ABB RAPID module: Module1.mod

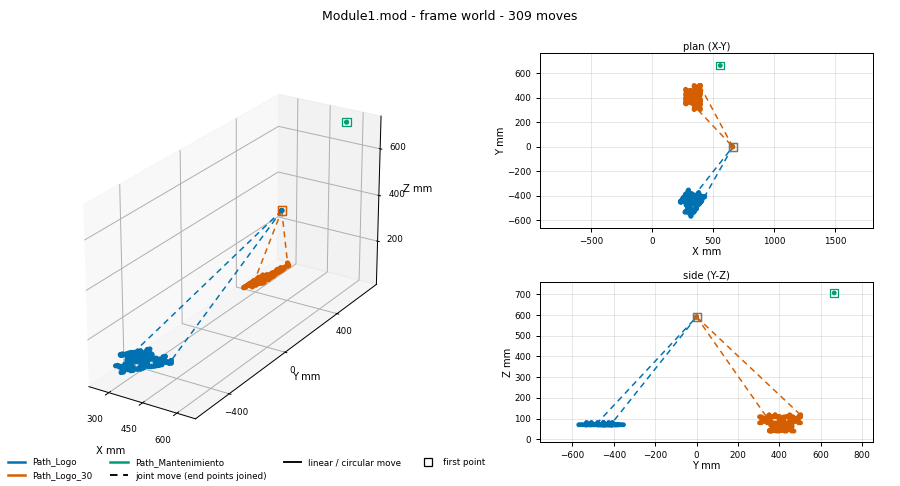
[picture p0: tool path of Module1.mod in frame world, 309 of 309 moves have a stored position in this frame; points joined in program order, loops and branches not executed]
MODULE Module1
        PERS tooldata TToolLab1:=[TRUE,[[120.208,0,145.208],[0.923879533,0,0.382683432,0]],[0.1,[47.87,0,69.665],[1,0,0,0],0,0,0]];
    TASK PERS wobjdata Logo:=[FALSE,TRUE,"",[[0,0,0],[1,0,0,0]],[[400,-450,60],[0.30070845,0,0,0.953716115]]];
    TASK PERS wobjdata Logo30:=[FALSE,TRUE,"",[[0,0,0],[1,0,0,0]],[[400,450,100],[0,-0.258819045,0,0.965925826]]];
    CONST robtarget Inicio:=[[44.962359667,-517.867347375,530.792],[0.115076142,0.881118798,0.277818382,-0.364971357],[0,0,-1,1],[9E+09,9E+09,9E+09,9E+09,9E+09,9E+09]];
    CONST robtarget X1_offset:=[[0,-52.582,20],[0,0,1,0],[-1,-3,-1,1],[9E+09,9E+09,9E+09,9E+09,9E+09,9E+09]];
    CONST robtarget Target_10:=[[0,-52.582,10],[0,0,1,0],[-1,-3,-1,1],[9E+09,9E+09,9E+09,9E+09,9E+09,9E+09]];
    CONST robtarget Target_20:=[[14.731,-43.214,10],[0,0,1,0],[-1,-3,-1,1],[9E+09,9E+09,9E+09,9E+09,9E+09,9E+09]];
    CONST robtarget Target_30:=[[29.461,-33.847,10],[0,0,1,0],[-1,-3,-1,1],[9E+09,9E+09,9E+09,9E+09,9E+09,9E+09]];
    CONST robtarget Target_40:=[[44.144,-42.928,10],[0,0,1,0],[-1,-3,-1,1],[9E+09,9E+09,9E+09,9E+09,9E+09,9E+09]];
    CONST robtarget Target_50:=[[58.827,-52.009,10],[0,0,1,0],[-1,-3,-1,1],[9E+09,9E+09,9E+09,9E+09,9E+09,9E+09]];
    CONST robtarget Target_60:=[[58.827,-43.047,10],[0,0,1,0],[-1,-3,-1,1],[9E+09,9E+09,9E+09,9E+09,9E+09,9E+09]];
    CONST robtarget Target_70:=[[47.314,-36.04,10],[0,0,1,0],[-1,-3,-1,1],[9E+09,9E+09,9E+09,9E+09,9E+09,9E+09]];
    CONST robtarget Target_80:=[[35.801,-29.032,10],[0,0,1,0],[-1,-3,-1,1],[9E+09,9E+09,9E+09,9E+09,9E+09,9E+09]];
    CONST robtarget Target_90:=[[47.314,-21.881,10],[0,0,1,0],[-1,-3,-1,1],[9E+09,9E+09,9E+09,9E+09,9E+09,9E+09]];
    CONST robtarget Target_100:=[[58.827,-14.73,10],[0,0,1,0],[-1,-3,-1,1],[9E+09,9E+09,9E+09,9E+09,9E+09,9E+09]];
    CONST robtarget Target_110:=[[58.827,-6.293,10],[0,0,1,0],[-1,-3,-1,1],[9E+09,9E+09,9E+09,9E+09,9E+09,9E+09]];
    CONST robtarget Target_120:=[[44.334,-15.493,10],[0,0,1,0],[-1,-3,-1,1],[9E+09,9E+09,9E+09,9E+09,9E+09,9E+09]];
    CONST robtarget Target_130:=[[29.842,-24.694,10],[0,0,1,0],[-1,-3,-1,1],[9E+09,9E+09,9E+09,9E+09,9E+09,9E+09]];
    CONST robtarget Target_140:=[[14.921,-15.493,10],[0,0,1,0],[-1,-3,-1,1],[9E+09,9E+09,9E+09,9E+09,9E+09,9E+09]];
    CONST robtarget Target_150:=[[0,-6.293,10],[0,0,1,0],[-1,-3,-1,1],[9E+09,9E+09,9E+09,9E+09,9E+09,9E+09]];
    CONST robtarget Target_160:=[[0,-15.255,10],[0,0,1,0],[-1,-3,-1,1],[9E+09,9E+09,9E+09,9E+09,9E+09,9E+09]];
    CONST robtarget Target_170:=[[11.727,-22.406,10],[0,0,1,0],[-1,-3,-1,1],[9E+09,9E+09,9E+09,9E+09,9E+09,9E+09]];
    CONST robtarget Target_180:=[[23.455,-29.556,10],[0,0,1,0],[-1,-3,-1,1],[9E+09,9E+09,9E+09,9E+09,9E+09,9E+09]];
    CONST robtarget Target_190:=[[11.727,-36.85,10],[0,0,1,0],[-1,-3,-1,1],[9E+09,9E+09,9E+09,9E+09,9E+09,9E+09]];
    CONST robtarget Target_200:=[[0,-44.144,10],[0,0,1,0],[-1,-3,-1,1],[9E+09,9E+09,9E+09,9E+09,9E+09,9E+09]];
    CONST robtarget B_offset:=[[0,0,20],[0,0,1,0],[-1,-3,-1,1],[9E+09,9E+09,9E+09,9E+09,9E+09,9E+09]];
    CONST robtarget Target_210:=[[0.000068234,0,10],[0,0,1,0],[-1,-3,-1,1],[9E+09,9E+09,9E+09,9E+09,9E+09,9E+09]];
    CONST robtarget Target_220:=[[29.413525648,0.000000006,10],[0,0,1,0],[-1,-3,-1,1],[9E+09,9E+09,9E+09,9E+09,9E+09,9E+09]];
    CONST robtarget Target_230:=[[58.826983061,0.000000012,10],[0,0,1,0],[-1,-3,-1,1],[9E+09,9E+09,9E+09,9E+09,9E+09,9E+09]];
    CONST robtarget Target_240:=[[58.826263831,7.794172482,10],[0,0,1,0],[-1,-3,-1,1],[9E+09,9E+09,9E+09,9E+09,9E+09,9E+09]];
    CONST robtarget Target_250:=[[58.826363749,15.588918532,10],[0,0,1,0],[-1,-3,-1,1],[9E+09,9E+09,9E+09,9E+09,9E+09,9E+09]];
    CONST robtarget Target_260:=[[58.421279237,25.027558611,10],[0,0,1,0],[-1,-3,-1,1],[9E+09,9E+09,9E+09,9E+09,9E+09,9E+09]];
    CONST robtarget Target_270:=[[56.442373859,31.03371666,10],[0,0,1,0],[-1,-3,-1,1],[9E+09,9E+09,9E+09,9E+09,9E+09,9E+09]];
    CONST robtarget Target_280:=[[52.032676311,35.682055346,10],[0,0,1,0],[-1,-3,-1,1],[9E+09,9E+09,9E+09,9E+09,9E+09,9E+09]];
    CONST robtarget Target_290:=[[45.573477335,37.136157676,10],[0,0,1,0],[-1,-3,-1,1],[9E+09,9E+09,9E+09,9E+09,9E+09,9E+09]];
    CONST robtarget Target_300:=[[38.136561779,34.942815929,10],[0,0,1,0],[-1,-3,-1,1],[9E+09,9E+09,9E+09,9E+09,9E+09,9E+09]];
    CONST robtarget Target_310:=[[32.98791054,28.888765515,10],[0,0,1,0],[-1,-3,-1,1],[9E+09,9E+09,9E+09,9E+09,9E+09,9E+09]];
    CONST robtarget Target_320:=[[27.482150174,37.016714998,10],[0,0,1,0],[-1,-3,-1,1],[9E+09,9E+09,9E+09,9E+09,9E+09,9E+09]];
    CONST robtarget Target_330:=[[18.067037183,39.901013935,10],[0,0,1,0],[-1,-3,-1,1],[9E+09,9E+09,9E+09,9E+09,9E+09,9E+09]];
    CONST robtarget Target_340:=[[10.320457963,38.231853851,10],[0,0,1,0],[-1,-3,-1,1],[9E+09,9E+09,9E+09,9E+09,9E+09,9E+09]];
    CONST robtarget Target_350:=[[4.766871396,33.798677084,10],[0,0,1,0],[-1,-3,-1,1],[9E+09,9E+09,9E+09,9E+09,9E+09,9E+09]];
    CONST robtarget Target_360:=[[1.096188095,26.671237284,10],[0,0,1,0],[-1,-3,-1,1],[9E+09,9E+09,9E+09,9E+09,9E+09,9E+09]];
    CONST robtarget Target_370:=[[-0.000000003,16.874785035,10],[0,0,1,0],[-1,-3,-1,1],[9E+09,9E+09,9E+09,9E+09,9E+09,9E+09]];
    CONST robtarget Target_380:=[[0.000156899,8.438088883,10],[0,0,1,0],[-1,-3,-1,1],[9E+09,9E+09,9E+09,9E+09,9E+09,9E+09]];
    CONST robtarget O_offset:=[[-1.24,70.315,20],[0,0,1,0],[-1,-3,-1,1],[9E+09,9E+09,9E+09,9E+09,9E+09,9E+09]];
    CONST robtarget Target_390:=[[-1.239782829,70.315479984,10],[0,0,1,0],[-1,-3,-1,1],[9E+09,9E+09,9E+09,9E+09,9E+09,9E+09]];
    CONST robtarget Target_400:=[[0.786338624,59.588668628,10],[0,0,1,0],[-1,-3,-1,1],[9E+09,9E+09,9E+09,9E+09,9E+09,9E+09]];
    CONST robtarget Target_410:=[[6.769482618,51.342081579,10],[0,0,1,0],[-1,-3,-1,1],[9E+09,9E+09,9E+09,9E+09,9E+09,9E+09]];
    CONST robtarget Target_420:=[[16.422507661,46.146190366,10],[0,0,1,0],[-1,-3,-1,1],[9E+09,9E+09,9E+09,9E+09,9E+09,9E+09]];
    CONST robtarget Target_430:=[[29.412921119,44.334619996,10],[0,0,1,0],[-1,-3,-1,1],[9E+09,9E+09,9E+09,9E+09,9E+09,9E+09]];
    CONST robtarget Target_440:=[[42.42730153,46.169208644,10],[0,0,1,0],[-1,-3,-1,1],[9E+09,9E+09,9E+09,9E+09,9E+09,9E+09]];
    CONST robtarget Target_450:=[[52.103968369,51.389690987,10],[0,0,1,0],[-1,-3,-1,1],[9E+09,9E+09,9E+09,9E+09,9E+09,9E+09]];
    CONST robtarget Target_460:=[[58.039423406,59.613427273,10],[0,0,1,0],[-1,-3,-1,1],[9E+09,9E+09,9E+09,9E+09,9E+09,9E+09]];
    CONST robtarget Target_470:=[[60.065636343,70.315019731,10],[0,0,1,0],[-1,-3,-1,1],[9E+09,9E+09,9E+09,9E+09,9E+09,9E+09]];
    CONST robtarget Target_480:=[[57.967982157,81.137015477,10],[0,0,1,0],[-1,-3,-1,1],[9E+09,9E+09,9E+09,9E+09,9E+09,9E+09]];
    CONST robtarget Target_490:=[[52.104377969,89.287851626,10],[0,0,1,0],[-1,-3,-1,1],[9E+09,9E+09,9E+09,9E+09,9E+09,9E+09]];
    CONST robtarget Target_500:=[[42.475192456,94.484565525,10],[0,0,1,0],[-1,-3,-1,1],[9E+09,9E+09,9E+09,9E+09,9E+09,9E+09]];
    CONST robtarget Target_510:=[[29.412679756,96.343313211,10],[0,0,1,0],[-1,-3,-1,1],[9E+09,9E+09,9E+09,9E+09,9E+09,9E+09]];
    CONST robtarget Target_520:=[[16.469896844,94.532001119,10],[0,0,1,0],[-1,-3,-1,1],[9E+09,9E+09,9E+09,9E+09,9E+09,9E+09]];
    CONST robtarget Target_530:=[[6.769065997,89.288494859,10],[0,0,1,0],[-1,-3,-1,1],[9E+09,9E+09,9E+09,9E+09,9E+09,9E+09]];
    CONST robtarget Target_540:=[[0.714522275,80.873942209,10],[0,0,1,0],[-1,-3,-1,1],[9E+09,9E+09,9E+09,9E+09,9E+09,9E+09]];
    CONST robtarget X2_offset:=[[0,99.299,20],[0,0,1,0],[-1,-3,-1,1],[9E+09,9E+09,9E+09,9E+09,9E+09,9E+09]];
    CONST robtarget Target_550:=[[0,99.299,10],[0,0,1,0],[-1,-3,-1,1],[9E+09,9E+09,9E+09,9E+09,9E+09,9E+09]];
    CONST robtarget Target_560:=[[14.73,108.667,10],[0,0,1,0],[-1,-3,-1,1],[9E+09,9E+09,9E+09,9E+09,9E+09,9E+09]];
    CONST robtarget Target_570:=[[29.46,118.034,10],[0,0,1,0],[-1,-3,-1,1],[9E+09,9E+09,9E+09,9E+09,9E+09,9E+09]];
    CONST robtarget Target_580:=[[44.143,108.953,10],[0,0,1,0],[-1,-3,-1,1],[9E+09,9E+09,9E+09,9E+09,9E+09,9E+09]];
    CONST robtarget Target_590:=[[58.826,99.871,10],[0,0,1,0],[-1,-3,-1,1],[9E+09,9E+09,9E+09,9E+09,9E+09,9E+09]];
    CONST robtarget Target_600:=[[58.826,108.834,10],[0,0,1,0],[-1,-3,-1,1],[9E+09,9E+09,9E+09,9E+09,9E+09,9E+09]];
    CONST robtarget Target_610:=[[47.313,115.841,10],[0,0,1,0],[-1,-3,-1,1],[9E+09,9E+09,9E+09,9E+09,9E+09,9E+09]];
    CONST robtarget Target_620:=[[35.801,122.849,10],[0,0,1,0],[-1,-3,-1,1],[9E+09,9E+09,9E+09,9E+09,9E+09,9E+09]];
    CONST robtarget Target_630:=[[47.313,130,10],[0,0,1,0],[-1,-3,-1,1],[9E+09,9E+09,9E+09,9E+09,9E+09,9E+09]];
    CONST robtarget Target_640:=[[58.826,137.15,10],[0,0,1,0],[-1,-3,-1,1],[9E+09,9E+09,9E+09,9E+09,9E+09,9E+09]];
    CONST robtarget Target_650:=[[58.826,145.588,10],[0,0,1,0],[-1,-3,-1,1],[9E+09,9E+09,9E+09,9E+09,9E+09,9E+09]];
    CONST robtarget Target_660:=[[44.334,136.388,10],[0,0,1,0],[-1,-3,-1,1],[9E+09,9E+09,9E+09,9E+09,9E+09,9E+09]];
    CONST robtarget Target_670:=[[29.842,127.187,10],[0,0,1,0],[-1,-3,-1,1],[9E+09,9E+09,9E+09,9E+09,9E+09,9E+09]];
    CONST robtarget Target_680:=[[14.92,136.387,10],[0,0,1,0],[-1,-3,-1,1],[9E+09,9E+09,9E+09,9E+09,9E+09,9E+09]];
    CONST robtarget Target_690:=[[-0.001,145.588,10],[0,0,1,0],[-1,-3,-1,1],[9E+09,9E+09,9E+09,9E+09,9E+09,9E+09]];
    CONST robtarget Target_700:=[[-0.001,136.626,10],[0,0,1,0],[-1,-3,-1,1],[9E+09,9E+09,9E+09,9E+09,9E+09,9E+09]];
    CONST robtarget Target_710:=[[11.726,129.475,10],[0,0,1,0],[-1,-3,-1,1],[9E+09,9E+09,9E+09,9E+09,9E+09,9E+09]];
    CONST robtarget Target_720:=[[23.454,122.324,10],[0,0,1,0],[-1,-3,-1,1],[9E+09,9E+09,9E+09,9E+09,9E+09,9E+09]];
    CONST robtarget Target_730:=[[11.727,115.031,10],[0,0,1,0],[-1,-3,-1,1],[9E+09,9E+09,9E+09,9E+09,9E+09,9E+09]];
    CONST robtarget Target_740:=[[-0.001,107.737,10],[0,0,1,0],[-1,-3,-1,1],[9E+09,9E+09,9E+09,9E+09,9E+09,9E+09]];
    CONST robtarget R_offset:=[[80.066,24.872,20],[0,0,1,0],[-1,-3,-1,1],[9E+09,9E+09,9E+09,9E+09,9E+09,9E+09]];
    CONST robtarget Target_750:=[[80.066,24.872,10],[0,0,1,0],[-1,-3,-1,1],[9E+09,9E+09,9E+09,9E+09,9E+09,9E+09]];
    CONST robtarget Target_760:=[[80.066,17.292,10],[0,0,1,0],[-1,-3,-1,1],[9E+09,9E+09,9E+09,9E+09,9E+09,9E+09]];
    CONST robtarget Target_770:=[[80.066,9.712,10],[0,0,1,0],[-1,-3,-1,1],[9E+09,9E+09,9E+09,9E+09,9E+09,9E+09]];
    CONST robtarget Target_780:=[[80.614,1.251,10],[0,0,1,0],[-1,-3,-1,1],[9E+09,9E+09,9E+09,9E+09,9E+09,9E+09]];
    CONST robtarget Target_790:=[[83.165,-5.256,10],[0,0,1,0],[-1,-3,-1,1],[9E+09,9E+09,9E+09,9E+09,9E+09,9E+09]];
    CONST robtarget Target_800:=[[88.289,-10.143,10],[0,0,1,0],[-1,-3,-1,1],[9E+09,9E+09,9E+09,9E+09,9E+09,9E+09]];
    CONST robtarget Target_810:=[[96.036,-11.93,10],[0,0,1,0],[-1,-3,-1,1],[9E+09,9E+09,9E+09,9E+09,9E+09,9E+09]];
    CONST robtarget Target_820:=[[106.833,-8.641,10],[0,0,1,0],[-1,-3,-1,1],[9E+09,9E+09,9E+09,9E+09,9E+09,9E+09]];
    CONST robtarget Target_830:=[[113.293,0.274,10],[0,0,1,0],[-1,-3,-1,1],[9E+09,9E+09,9E+09,9E+09,9E+09,9E+09]];
    CONST robtarget Target_840:=[[126.093,-10.19,10],[0,0,1,0],[-1,-3,-1,1],[9E+09,9E+09,9E+09,9E+09,9E+09,9E+09]];
    CONST robtarget Target_850:=[[138.892,-20.654,10],[0,0,1,0],[-1,-3,-1,1],[9E+09,9E+09,9E+09,9E+09,9E+09,9E+09]];
    CONST robtarget Target_860:=[[138.892,-10.5,10],[0,0,1,0],[-1,-3,-1,1],[9E+09,9E+09,9E+09,9E+09,9E+09,9E+09]];
    CONST robtarget Target_870:=[[127.189,-1.204,10],[0,0,1,0],[-1,-3,-1,1],[9E+09,9E+09,9E+09,9E+09,9E+09,9E+09]];
    CONST robtarget Target_880:=[[115.486,8.092,10],[0,0,1,0],[-1,-3,-1,1],[9E+09,9E+09,9E+09,9E+09,9E+09,9E+09]];
    CONST robtarget Target_890:=[[115.486,17.054,10],[0,0,1,0],[-1,-3,-1,1],[9E+09,9E+09,9E+09,9E+09,9E+09,9E+09]];
    CONST robtarget Target_900:=[[127.189,17.054,10],[0,0,1,0],[-1,-3,-1,1],[9E+09,9E+09,9E+09,9E+09,9E+09,9E+09]];
    CONST robtarget Target_910:=[[138.892,17.054,10],[0,0,1,0],[-1,-3,-1,1],[9E+09,9E+09,9E+09,9E+09,9E+09,9E+09]];
    CONST robtarget Target_920:=[[138.892,24.872,10],[0,0,1,0],[-1,-3,-1,1],[9E+09,9E+09,9E+09,9E+09,9E+09,9E+09]];
    CONST robtarget Target_930:=[[109.479,24.872,10],[0,0,1,0],[-1,-3,-1,1],[9E+09,9E+09,9E+09,9E+09,9E+09,9E+09]];
    CONST robtarget J1_offset:=[[80.066,56.669,20],[0,0,1,0],[-1,-3,-1,1],[9E+09,9E+09,9E+09,9E+09,9E+09,9E+09]];
    CONST robtarget Target_940:=[[80.066,56.669,10],[0,0,1,0],[-1,-3,-1,1],[9E+09,9E+09,9E+09,9E+09,9E+09,9E+09]];
    CONST robtarget Target_950:=[[80.066,46.538,10],[0,0,1,0],[-1,-3,-1,1],[9E+09,9E+09,9E+09,9E+09,9E+09,9E+09]];
    CONST robtarget Target_960:=[[80.066,36.408,10],[0,0,1,0],[-1,-3,-1,1],[9E+09,9E+09,9E+09,9E+09,9E+09,9E+09]];
    CONST robtarget Target_970:=[[101.828,36.408,10],[0,0,1,0],[-1,-3,-1,1],[9E+09,9E+09,9E+09,9E+09,9E+09,9E+09]];
    CONST robtarget Target_980:=[[123.59,36.408,10],[0,0,1,0],[-1,-3,-1,1],[9E+09,9E+09,9E+09,9E+09,9E+09,9E+09]];
    CONST robtarget Target_990:=[[135.507,41.128,10],[0,0,1,0],[-1,-3,-1,1],[9E+09,9E+09,9E+09,9E+09,9E+09,9E+09]];
    CONST robtarget Target_1000:=[[139.702,53.809,10],[0,0,1,0],[-1,-3,-1,1],[9E+09,9E+09,9E+09,9E+09,9E+09,9E+09]];
    CONST robtarget Target_1010:=[[138.558,64.201,10],[0,0,1,0],[-1,-3,-1,1],[9E+09,9E+09,9E+09,9E+09,9E+09,9E+09]];
    CONST robtarget Target_1020:=[[131.026,63.772,10],[0,0,1,0],[-1,-3,-1,1],[9E+09,9E+09,9E+09,9E+09,9E+09,9E+09]];
    CONST robtarget Target_1030:=[[132.266,59.744,10],[0,0,1,0],[-1,-3,-1,1],[9E+09,9E+09,9E+09,9E+09,9E+09,9E+09]];
    CONST robtarget Target_1040:=[[132.933,54.857,10],[0,0,1,0],[-1,-3,-1,1],[9E+09,9E+09,9E+09,9E+09,9E+09,9E+09]];
    CONST robtarget Target_1050:=[[132.099,49.065,10],[0,0,1,0],[-1,-3,-1,1],[9E+09,9E+09,9E+09,9E+09,9E+09,9E+09]];
    CONST robtarget Target_1060:=[[129.739,45.895,10],[0,0,1,0],[-1,-3,-1,1],[9E+09,9E+09,9E+09,9E+09,9E+09,9E+09]];
    CONST robtarget Target_1070:=[[125.878,44.513,10],[0,0,1,0],[-1,-3,-1,1],[9E+09,9E+09,9E+09,9E+09,9E+09,9E+09]];
    CONST robtarget Target_1080:=[[120.586,44.227,10],[0,0,1,0],[-1,-3,-1,1],[9E+09,9E+09,9E+09,9E+09,9E+09,9E+09]];
    CONST robtarget Target_1090:=[[103.448,44.226,10],[0,0,1,0],[-1,-3,-1,1],[9E+09,9E+09,9E+09,9E+09,9E+09,9E+09]];
    CONST robtarget Target_1100:=[[86.311,44.226,10],[0,0,1,0],[-1,-3,-1,1],[9E+09,9E+09,9E+09,9E+09,9E+09,9E+09]];
    CONST robtarget Target_1110:=[[86.311,56.669,10],[0,0,1,0],[-1,-3,-1,1],[9E+09,9E+09,9E+09,9E+09,9E+09,9E+09]];
    CONST robtarget J2_offset:=[[80.065,90.372,20],[0,0,1,0],[-1,-3,-1,1],[9E+09,9E+09,9E+09,9E+09,9E+09,9E+09]];
    CONST robtarget Target_1120:=[[80.065,90.372,10],[0,0,1,0],[-1,-3,-1,1],[9E+09,9E+09,9E+09,9E+09,9E+09,9E+09]];
    CONST robtarget Target_1130:=[[80.065,80.242,10],[0,0,1,0],[-1,-3,-1,1],[9E+09,9E+09,9E+09,9E+09,9E+09,9E+09]];
    CONST robtarget Target_1140:=[[80.066,70.112,10],[0,0,1,0],[-1,-3,-1,1],[9E+09,9E+09,9E+09,9E+09,9E+09,9E+09]];
    CONST robtarget Target_1150:=[[101.827,70.112,10],[0,0,1,0],[-1,-3,-1,1],[9E+09,9E+09,9E+09,9E+09,9E+09,9E+09]];
    CONST robtarget Target_1160:=[[123.589,70.112,10],[0,0,1,0],[-1,-3,-1,1],[9E+09,9E+09,9E+09,9E+09,9E+09,9E+09]];
    CONST robtarget Target_1170:=[[135.507,74.832,10],[0,0,1,0],[-1,-3,-1,1],[9E+09,9E+09,9E+09,9E+09,9E+09,9E+09]];
    CONST robtarget Target_1180:=[[139.702,87.512,10],[0,0,1,0],[-1,-3,-1,1],[9E+09,9E+09,9E+09,9E+09,9E+09,9E+09]];
    CONST robtarget Target_1190:=[[139.369,92.589,10],[0,0,1,0],[-1,-3,-1,1],[9E+09,9E+09,9E+09,9E+09,9E+09,9E+09]];
    CONST robtarget Target_1200:=[[138.558,97.905,10],[0,0,1,0],[-1,-3,-1,1],[9E+09,9E+09,9E+09,9E+09,9E+09,9E+09]];
    CONST robtarget Target_1210:=[[134.792,97.905,10],[0,0,1,0],[-1,-3,-1,1],[9E+09,9E+09,9E+09,9E+09,9E+09,9E+09]];
    CONST robtarget Target_1220:=[[131.026,97.475,10],[0,0,1,0],[-1,-3,-1,1],[9E+09,9E+09,9E+09,9E+09,9E+09,9E+09]];
    CONST robtarget Target_1230:=[[132.265,93.447,10],[0,0,1,0],[-1,-3,-1,1],[9E+09,9E+09,9E+09,9E+09,9E+09,9E+09]];
    CONST robtarget Target_1240:=[[132.933,88.561,10],[0,0,1,0],[-1,-3,-1,1],[9E+09,9E+09,9E+09,9E+09,9E+09,9E+09]];
    CONST robtarget Target_1250:=[[132.099,82.769,10],[0,0,1,0],[-1,-3,-1,1],[9E+09,9E+09,9E+09,9E+09,9E+09,9E+09]];
    CONST robtarget Target_1260:=[[129.739,79.599,10],[0,0,1,0],[-1,-3,-1,1],[9E+09,9E+09,9E+09,9E+09,9E+09,9E+09]];
    CONST robtarget Target_1270:=[[125.878,78.216,10],[0,0,1,0],[-1,-3,-1,1],[9E+09,9E+09,9E+09,9E+09,9E+09,9E+09]];
    CONST robtarget Target_1280:=[[120.586,77.93,10],[0,0,1,0],[-1,-3,-1,1],[9E+09,9E+09,9E+09,9E+09,9E+09,9E+09]];
    CONST robtarget Target_1290:=[[110.666,78.402,10],[0,0,1,0],[-1,-3,-1,1],[9E+09,9E+09,9E+09,9E+09,9E+09,9E+09]];
    CONST robtarget Target_1300:=[[86.31,77.93,10],[0,0,1,0],[-1,-3,-1,1],[9E+09,9E+09,9E+09,9E+09,9E+09,9E+09]];
    CONST robtarget Target_1310:=[[86.31,90.372,10],[0,0,1,0],[-1,-3,-1,1],[9E+09,9E+09,9E+09,9E+09,9E+09,9E+09]];
    CONST robtarget Circle_offset:=[[-40.933895973,-5.82304871,40],[0,1,0,0],[-1,-1,0,1],[9E+09,9E+09,9E+09,9E+09,9E+09,9E+09]];
    CONST robtarget Target_1330:=[[-40.933895973,-5.82304871,10],[0,1,0,0],[-1,-1,0,1],[9E+09,9E+09,9E+09,9E+09,9E+09,9E+09]];
    CONST robtarget Target_1340:=[[-19.93416425,39.773116891,10],[0,1,0,0],[-1,-1,0,1],[9E+09,9E+09,9E+09,9E+09,9E+09,9E+09]];
    CONST robtarget Target_1350:=[[-40.934569392,85.369917227,10],[0,1,0,0],[-1,-1,0,1],[9E+09,9E+09,9E+09,9E+09,9E+09,9E+09]];
    CONST robtarget Target_1360:=[[-45.307466947,88.773192557,10],[0,1,0,0],[-1,-1,0,1],[9E+09,9E+09,9E+09,9E+09,9E+09,9E+09]];
    CONST robtarget Target_1370:=[[-86.904601275,99.366718349,10],[0,1,0,0],[-1,-1,0,1],[9E+09,9E+09,9E+09,9E+09,9E+09,9E+09]];
    CONST robtarget Target_1380:=[[-124.934724159,79.459035651,10],[0,1,0,0],[-1,-1,0,1],[9E+09,9E+09,9E+09,9E+09,9E+09,9E+09]];
    CONST robtarget Target_1390:=[[-132.460361347,68.772867492,10],[0,1,0,0],[-1,-1,0,1],[9E+09,9E+09,9E+09,9E+09,9E+09,9E+09]];
    CONST robtarget Target_1400:=[[-139.934438017,39.773268565,10],[0,1,0,0],[-1,-1,0,1],[9E+09,9E+09,9E+09,9E+09,9E+09,9E+09]];
    CONST robtarget Target_1410:=[[-132.460399107,10.77239383,10],[0,1,0,0],[-1,-1,0,1],[9E+09,9E+09,9E+09,9E+09,9E+09,9E+09]];
    CONST robtarget Target_1420:=[[-124.934206216,0.086767195,10],[0,1,0,0],[-1,-1,0,1],[9E+09,9E+09,9E+09,9E+09,9E+09,9E+09]];
    CONST robtarget Target_1430:=[[-86.904215372,-19.820139957,10],[0,1,0,0],[-1,-1,0,1],[9E+09,9E+09,9E+09,9E+09,9E+09,9E+09]];
    CONST robtarget Target_1440:=[[-45.307855796,-9.226362018,10],[0,1,0,0],[-1,-1,0,1],[9E+09,9E+09,9E+09,9E+09,9E+09,9E+09]];
    CONST robtarget Target_1450:=[[-80.972940534,2.559268073,10],[0,1,0,0],[-1,-1,0,1],[9E+09,9E+09,9E+09,9E+09,9E+09,9E+09]];
    CONST robtarget Target_1460:=[[-110.207862361,26.143998086,10],[0,1,0,0],[-1,-1,0,1],[9E+09,9E+09,9E+09,9E+09,9E+09,9E+09]];
    CONST robtarget Target_1470:=[[-118.12963234,13.431074685,10],[0,1,0,0],[-1,-1,0,1],[9E+09,9E+09,9E+09,9E+09,9E+09,9E+09]];
    CONST robtarget Target_1480:=[[-124.934206216,0.086767195,10],[0,1,0,0],[-1,-1,0,1],[9E+09,9E+09,9E+09,9E+09,9E+09,9E+09]];
    CONST robtarget Target_1490:=[[-132.460399107,10.77239383,10],[0,1,0,0],[-1,-1,0,1],[9E+09,9E+09,9E+09,9E+09,9E+09,9E+09]];
    CONST robtarget Target_1500:=[[-127.413721906,25.736314013,10],[0,1,0,0],[-1,-1,0,1],[9E+09,9E+09,9E+09,9E+09,9E+09,9E+09]];
    CONST robtarget Target_1510:=[[-120.179725035,39.773180446,10],[0,1,0,0],[-1,-1,0,1],[9E+09,9E+09,9E+09,9E+09,9E+09,9E+09]];
    CONST robtarget Target_1520:=[[-127.413036308,53.809835782,10],[0,1,0,0],[-1,-1,0,1],[9E+09,9E+09,9E+09,9E+09,9E+09,9E+09]];
    CONST robtarget Target_1530:=[[-132.460361347,68.772867492,10],[0,1,0,0],[-1,-1,0,1],[9E+09,9E+09,9E+09,9E+09,9E+09,9E+09]];
    CONST robtarget Target_1540:=[[-124.934724159,79.459035651,10],[0,1,0,0],[-1,-1,0,1],[9E+09,9E+09,9E+09,9E+09,9E+09,9E+09]];
    CONST robtarget Target_1550:=[[-118.129234234,66.115306641,10],[0,1,0,0],[-1,-1,0,1],[9E+09,9E+09,9E+09,9E+09,9E+09,9E+09]];
    CONST robtarget Target_1560:=[[-110.208779056,53.402138084,10],[0,1,0,0],[-1,-1,0,1],[9E+09,9E+09,9E+09,9E+09,9E+09,9E+09]];
    CONST robtarget Target_1570:=[[-80.973561626,76.987307975,10],[0,1,0,0],[-1,-1,0,1],[9E+09,9E+09,9E+09,9E+09,9E+09,9E+09]];
    CONST robtarget Target_1580:=[[-45.307466947,88.773192557,10],[0,1,0,0],[-1,-1,0,1],[9E+09,9E+09,9E+09,9E+09,9E+09,9E+09]];
    CONST robtarget Target_1590:=[[-40.934569392,85.369917227,10],[0,1,0,0],[-1,-1,0,1],[9E+09,9E+09,9E+09,9E+09,9E+09,9E+09]];
    CONST robtarget Target_1600:=[[-72.858424166,65.74477085,10],[0,1,0,0],[-1,-1,0,1],[9E+09,9E+09,9E+09,9E+09,9E+09,9E+09]];
    CONST robtarget Target_1610:=[[-99.870719718,39.77300876,10],[0,1,0,0],[-1,-1,0,1],[9E+09,9E+09,9E+09,9E+09,9E+09,9E+09]];
    CONST robtarget Target_1620:=[[-72.85802852,13.802107751,10],[0,1,0,0],[-1,-1,0,1],[9E+09,9E+09,9E+09,9E+09,9E+09,9E+09]];
    CONST robtarget Target_1630:=[[-40.933895973,-5.82304871,10],[0,1,0,0],[-1,-1,0,1],[9E+09,9E+09,9E+09,9E+09,9E+09,9E+09]];
    CONST robtarget X1_offset_2:=[[0,-52.582,20],[0,0,1,0],[0,0,-2,0],[9E+09,9E+09,9E+09,9E+09,9E+09,9E+09]];
    CONST robtarget Target_10_2:=[[0,-52.582,10],[0,0,1,0],[0,0,-2,0],[9E+09,9E+09,9E+09,9E+09,9E+09,9E+09]];
    CONST robtarget Target_20_2:=[[14.731,-43.214,10],[0,0,1,0],[0,0,-2,0],[9E+09,9E+09,9E+09,9E+09,9E+09,9E+09]];
    CONST robtarget Target_30_2:=[[29.461,-33.847,10],[0,0,1,0],[0,0,-2,0],[9E+09,9E+09,9E+09,9E+09,9E+09,9E+09]];
    CONST robtarget Target_40_2:=[[44.144,-42.928,10],[0,0,1,0],[0,0,-2,0],[9E+09,9E+09,9E+09,9E+09,9E+09,9E+09]];
    CONST robtarget Target_50_2:=[[58.827,-52.009,10],[0,0,1,0],[0,0,-2,0],[9E+09,9E+09,9E+09,9E+09,9E+09,9E+09]];
    CONST robtarget Target_60_2:=[[58.827,-43.047,10],[0,0,1,0],[0,0,-2,0],[9E+09,9E+09,9E+09,9E+09,9E+09,9E+09]];
    CONST robtarget Target_70_2:=[[47.314,-36.04,10],[0,0,1,0],[0,0,-2,0],[9E+09,9E+09,9E+09,9E+09,9E+09,9E+09]];
    CONST robtarget Target_80_2:=[[35.801,-29.032,10],[0,0,1,0],[0,0,-2,0],[9E+09,9E+09,9E+09,9E+09,9E+09,9E+09]];
    CONST robtarget Target_90_2:=[[47.314,-21.881,10],[0,0,1,0],[0,0,-2,0],[9E+09,9E+09,9E+09,9E+09,9E+09,9E+09]];
    CONST robtarget Target_100_2:=[[58.827,-14.73,10],[0,0,1,0],[0,0,-2,0],[9E+09,9E+09,9E+09,9E+09,9E+09,9E+09]];
    CONST robtarget Target_110_2:=[[58.827,-6.293,10],[0,0,1,0],[0,0,-2,0],[9E+09,9E+09,9E+09,9E+09,9E+09,9E+09]];
    CONST robtarget Target_120_2:=[[44.334,-15.493,10],[0,0,1,0],[0,0,-2,0],[9E+09,9E+09,9E+09,9E+09,9E+09,9E+09]];
    CONST robtarget Target_130_2:=[[29.842,-24.694,10],[0,0,1,0],[0,0,-2,0],[9E+09,9E+09,9E+09,9E+09,9E+09,9E+09]];
    CONST robtarget Target_140_2:=[[14.921,-15.493,10],[0,0,1,0],[0,0,-2,0],[9E+09,9E+09,9E+09,9E+09,9E+09,9E+09]];
    CONST robtarget Target_150_2:=[[0,-6.293,10],[0,0,1,0],[0,0,-2,0],[9E+09,9E+09,9E+09,9E+09,9E+09,9E+09]];
    CONST robtarget Target_160_2:=[[0,-15.255,10],[0,0,1,0],[0,0,-2,0],[9E+09,9E+09,9E+09,9E+09,9E+09,9E+09]];
    CONST robtarget Target_170_2:=[[11.727,-22.406,10],[0,0,1,0],[0,0,-2,0],[9E+09,9E+09,9E+09,9E+09,9E+09,9E+09]];
    CONST robtarget Target_180_2:=[[23.455,-29.556,10],[0,0,1,0],[0,0,-2,0],[9E+09,9E+09,9E+09,9E+09,9E+09,9E+09]];
    CONST robtarget Target_190_2:=[[11.727,-36.85,10],[0,0,1,0],[0,0,-2,0],[9E+09,9E+09,9E+09,9E+09,9E+09,9E+09]];
    CONST robtarget Target_200_2:=[[0,-44.144,10],[0,0,1,0],[0,0,-2,0],[9E+09,9E+09,9E+09,9E+09,9E+09,9E+09]];
    CONST robtarget B_offset_2:=[[0,0,20],[0,0,1,0],[0,0,-2,0],[9E+09,9E+09,9E+09,9E+09,9E+09,9E+09]];
    CONST robtarget Target_210_2:=[[0.000068234,0,10],[0,0,1,0],[0,0,-2,0],[9E+09,9E+09,9E+09,9E+09,9E+09,9E+09]];
    CONST robtarget Target_220_2:=[[29.413525648,0.000000006,10],[0,0,1,0],[0,0,-2,0],[9E+09,9E+09,9E+09,9E+09,9E+09,9E+09]];
    CONST robtarget Target_230_2:=[[58.826983061,0.000000012,10],[0,0,1,0],[0,0,-2,0],[9E+09,9E+09,9E+09,9E+09,9E+09,9E+09]];
    CONST robtarget Target_240_2:=[[58.826263831,7.794172482,10],[0,0,1,0],[0,0,-2,0],[9E+09,9E+09,9E+09,9E+09,9E+09,9E+09]];
    CONST robtarget Target_250_2:=[[58.826363749,15.588918532,10],[0,0,1,0],[0,0,-2,0],[9E+09,9E+09,9E+09,9E+09,9E+09,9E+09]];
    CONST robtarget Target_260_2:=[[58.421279237,25.027558611,10],[0,0,1,0],[0,0,-2,0],[9E+09,9E+09,9E+09,9E+09,9E+09,9E+09]];
    CONST robtarget Target_270_2:=[[56.442373859,31.03371666,10],[0,0,1,0],[0,0,-2,0],[9E+09,9E+09,9E+09,9E+09,9E+09,9E+09]];
    CONST robtarget Target_280_2:=[[52.032676311,35.682055346,10],[0,0,1,0],[0,0,-2,0],[9E+09,9E+09,9E+09,9E+09,9E+09,9E+09]];
    CONST robtarget Target_290_2:=[[45.573477335,37.136157676,10],[0,0,1,0],[0,0,-2,0],[9E+09,9E+09,9E+09,9E+09,9E+09,9E+09]];
    CONST robtarget Target_300_2:=[[38.136561779,34.942815929,10],[0,0,1,0],[0,0,-2,0],[9E+09,9E+09,9E+09,9E+09,9E+09,9E+09]];
    CONST robtarget Target_310_2:=[[32.98791054,28.888765515,10],[0,0,1,0],[0,0,-2,0],[9E+09,9E+09,9E+09,9E+09,9E+09,9E+09]];
    CONST robtarget Target_320_2:=[[27.482150174,37.016714998,10],[0,0,1,0],[0,0,-2,0],[9E+09,9E+09,9E+09,9E+09,9E+09,9E+09]];
    CONST robtarget Target_330_2:=[[18.067037183,39.901013935,10],[0,0,1,0],[0,0,-2,0],[9E+09,9E+09,9E+09,9E+09,9E+09,9E+09]];
    CONST robtarget Target_340_2:=[[10.320457963,38.231853851,10],[0,0,1,0],[0,0,-2,0],[9E+09,9E+09,9E+09,9E+09,9E+09,9E+09]];
    CONST robtarget Target_350_2:=[[4.766871396,33.798677084,10],[0,0,1,0],[0,0,-2,0],[9E+09,9E+09,9E+09,9E+09,9E+09,9E+09]];
    CONST robtarget Target_360_2:=[[1.096188095,26.671237284,10],[0,0,1,0],[0,0,-2,0],[9E+09,9E+09,9E+09,9E+09,9E+09,9E+09]];
    CONST robtarget Target_370_2:=[[-0.000000003,16.874785035,10],[0,0,1,0],[0,0,-2,0],[9E+09,9E+09,9E+09,9E+09,9E+09,9E+09]];
    CONST robtarget Target_380_2:=[[0.000156899,8.438088883,10],[0,0,1,0],[0,0,-2,0],[9E+09,9E+09,9E+09,9E+09,9E+09,9E+09]];
    CONST robtarget O_offset_2:=[[-1.24,70.315,20],[0,0,1,0],[0,0,-2,0],[9E+09,9E+09,9E+09,9E+09,9E+09,9E+09]];
    CONST robtarget Target_390_2:=[[-1.239782829,70.315479984,10],[0,0,1,0],[0,0,-2,0],[9E+09,9E+09,9E+09,9E+09,9E+09,9E+09]];
    CONST robtarget Target_400_2:=[[0.786338624,59.588668628,10],[0,0,1,0],[0,0,-2,0],[9E+09,9E+09,9E+09,9E+09,9E+09,9E+09]];
    CONST robtarget Target_410_2:=[[6.769482618,51.342081579,10],[0,0,1,0],[0,0,-2,0],[9E+09,9E+09,9E+09,9E+09,9E+09,9E+09]];
    CONST robtarget Target_420_2:=[[16.422507661,46.146190366,10],[0,0,1,0],[0,0,-2,0],[9E+09,9E+09,9E+09,9E+09,9E+09,9E+09]];
    CONST robtarget Target_430_2:=[[29.412921119,44.334619996,10],[0,0,1,0],[0,0,-2,0],[9E+09,9E+09,9E+09,9E+09,9E+09,9E+09]];
    CONST robtarget Target_440_2:=[[42.42730153,46.169208644,10],[0,0,1,0],[0,0,-2,0],[9E+09,9E+09,9E+09,9E+09,9E+09,9E+09]];
    CONST robtarget Target_450_2:=[[52.103968369,51.389690987,10],[0,0,1,0],[0,0,-2,0],[9E+09,9E+09,9E+09,9E+09,9E+09,9E+09]];
    CONST robtarget Target_460_2:=[[58.039423406,59.613427273,10],[0,0,1,0],[0,0,-2,0],[9E+09,9E+09,9E+09,9E+09,9E+09,9E+09]];
    CONST robtarget Target_470_2:=[[60.065636343,70.315019731,10],[0,0,1,0],[0,0,-2,0],[9E+09,9E+09,9E+09,9E+09,9E+09,9E+09]];
    CONST robtarget Target_480_2:=[[57.967982157,81.137015477,10],[0,0,1,0],[0,0,-2,0],[9E+09,9E+09,9E+09,9E+09,9E+09,9E+09]];
    CONST robtarget Target_490_2:=[[52.104377969,89.287851626,10],[0,0,1,0],[0,0,-2,0],[9E+09,9E+09,9E+09,9E+09,9E+09,9E+09]];
    CONST robtarget Target_500_2:=[[42.475192456,94.484565525,10],[0,0,1,0],[0,0,-2,0],[9E+09,9E+09,9E+09,9E+09,9E+09,9E+09]];
    CONST robtarget Target_510_2:=[[29.412679756,96.343313211,10],[0,0,1,0],[0,0,-2,0],[9E+09,9E+09,9E+09,9E+09,9E+09,9E+09]];
    CONST robtarget Target_520_2:=[[16.469896844,94.532001119,10],[0,0,1,0],[0,0,-2,0],[9E+09,9E+09,9E+09,9E+09,9E+09,9E+09]];
    CONST robtarget Target_530_2:=[[6.769065997,89.288494859,10],[0,0,1,0],[0,0,-2,0],[9E+09,9E+09,9E+09,9E+09,9E+09,9E+09]];
    CONST robtarget Target_540_2:=[[0.714522275,80.873942209,10],[0,0,1,0],[0,0,-2,0],[9E+09,9E+09,9E+09,9E+09,9E+09,9E+09]];
    CONST robtarget X2_offset_2:=[[0,99.299,20],[0,0,1,0],[0,0,-2,0],[9E+09,9E+09,9E+09,9E+09,9E+09,9E+09]];
    CONST robtarget Target_550_2:=[[0,99.299,10],[0,0,1,0],[0,0,-2,0],[9E+09,9E+09,9E+09,9E+09,9E+09,9E+09]];
    CONST robtarget Target_560_2:=[[14.73,108.667,10],[0,0,1,0],[0,0,-2,0],[9E+09,9E+09,9E+09,9E+09,9E+09,9E+09]];
    CONST robtarget Target_570_2:=[[29.46,118.034,10],[0,0,1,0],[0,0,-2,0],[9E+09,9E+09,9E+09,9E+09,9E+09,9E+09]];
    CONST robtarget Target_580_2:=[[44.143,108.953,10],[0,0,1,0],[0,0,-2,0],[9E+09,9E+09,9E+09,9E+09,9E+09,9E+09]];
    CONST robtarget Target_590_2:=[[58.826,99.871,10],[0,0,1,0],[0,0,-2,0],[9E+09,9E+09,9E+09,9E+09,9E+09,9E+09]];
    CONST robtarget Target_600_2:=[[58.826,108.834,10],[0,0,1,0],[0,0,-2,0],[9E+09,9E+09,9E+09,9E+09,9E+09,9E+09]];
    CONST robtarget Target_610_2:=[[47.313,115.841,10],[0,0,1,0],[0,0,-2,0],[9E+09,9E+09,9E+09,9E+09,9E+09,9E+09]];
    CONST robtarget Target_620_2:=[[35.801,122.849,10],[0,0,1,0],[0,0,-2,0],[9E+09,9E+09,9E+09,9E+09,9E+09,9E+09]];
    CONST robtarget Target_630_2:=[[47.313,130,10],[0,0,1,0],[0,0,-2,0],[9E+09,9E+09,9E+09,9E+09,9E+09,9E+09]];
    CONST robtarget Target_640_2:=[[58.826,137.15,10],[0,0,1,0],[0,0,-2,0],[9E+09,9E+09,9E+09,9E+09,9E+09,9E+09]];
    CONST robtarget Target_650_2:=[[58.826,145.588,10],[0,0,1,0],[0,0,-2,0],[9E+09,9E+09,9E+09,9E+09,9E+09,9E+09]];
    CONST robtarget Target_660_2:=[[44.334,136.388,10],[0,0,1,0],[0,0,-2,0],[9E+09,9E+09,9E+09,9E+09,9E+09,9E+09]];
    CONST robtarget Target_670_2:=[[29.842,127.187,10],[0,0,1,0],[0,0,-2,0],[9E+09,9E+09,9E+09,9E+09,9E+09,9E+09]];
    CONST robtarget Target_680_2:=[[14.92,136.387,10],[0,0,1,0],[0,0,-2,0],[9E+09,9E+09,9E+09,9E+09,9E+09,9E+09]];
    CONST robtarget Target_690_2:=[[-0.001,145.588,10],[0,0,1,0],[0,0,-2,0],[9E+09,9E+09,9E+09,9E+09,9E+09,9E+09]];
    CONST robtarget Target_700_2:=[[-0.001,136.626,10],[0,0,1,0],[0,0,-2,0],[9E+09,9E+09,9E+09,9E+09,9E+09,9E+09]];
    CONST robtarget Target_710_2:=[[11.726,129.475,10],[0,0,1,0],[0,0,-2,0],[9E+09,9E+09,9E+09,9E+09,9E+09,9E+09]];
    CONST robtarget Target_720_2:=[[23.454,122.324,10],[0,0,1,0],[0,0,-2,0],[9E+09,9E+09,9E+09,9E+09,9E+09,9E+09]];
    CONST robtarget Target_730_2:=[[11.727,115.031,10],[0,0,1,0],[0,0,-2,0],[9E+09,9E+09,9E+09,9E+09,9E+09,9E+09]];
    CONST robtarget Target_740_2:=[[-0.001,107.737,10],[0,0,1,0],[0,0,-2,0],[9E+09,9E+09,9E+09,9E+09,9E+09,9E+09]];
    CONST robtarget R_offset_2:=[[80.066,24.872,20],[0,0,1,0],[0,0,-2,0],[9E+09,9E+09,9E+09,9E+09,9E+09,9E+09]];
    CONST robtarget Target_750_2:=[[80.066,24.872,10],[0,0,1,0],[0,0,-2,0],[9E+09,9E+09,9E+09,9E+09,9E+09,9E+09]];
    CONST robtarget Target_760_2:=[[80.066,17.292,10],[0,0,1,0],[0,0,-2,0],[9E+09,9E+09,9E+09,9E+09,9E+09,9E+09]];
    CONST robtarget Target_770_2:=[[80.066,9.712,10],[0,0,1,0],[0,0,-2,0],[9E+09,9E+09,9E+09,9E+09,9E+09,9E+09]];
    CONST robtarget Target_780_2:=[[80.614,1.251,10],[0,0,1,0],[0,0,-2,0],[9E+09,9E+09,9E+09,9E+09,9E+09,9E+09]];
    CONST robtarget Target_790_2:=[[83.165,-5.256,10],[0,0,1,0],[0,0,-2,0],[9E+09,9E+09,9E+09,9E+09,9E+09,9E+09]];
    CONST robtarget Target_800_2:=[[88.289,-10.143,10],[0,0,1,0],[0,0,-2,0],[9E+09,9E+09,9E+09,9E+09,9E+09,9E+09]];
    CONST robtarget Target_810_2:=[[96.036,-11.93,10],[0,0,1,0],[0,0,-2,0],[9E+09,9E+09,9E+09,9E+09,9E+09,9E+09]];
    CONST robtarget Target_820_2:=[[106.833,-8.641,10],[0,0,1,0],[0,0,-2,0],[9E+09,9E+09,9E+09,9E+09,9E+09,9E+09]];
    CONST robtarget Target_830_2:=[[113.293,0.274,10],[0,0,1,0],[0,0,-2,0],[9E+09,9E+09,9E+09,9E+09,9E+09,9E+09]];
    CONST robtarget Target_840_2:=[[126.093,-10.19,10],[0,0,1,0],[0,0,-2,0],[9E+09,9E+09,9E+09,9E+09,9E+09,9E+09]];
    CONST robtarget Target_850_2:=[[138.892,-20.654,10],[0,0,1,0],[0,0,-2,0],[9E+09,9E+09,9E+09,9E+09,9E+09,9E+09]];
    CONST robtarget Target_860_2:=[[138.892,-10.5,10],[0,0,1,0],[0,0,-2,0],[9E+09,9E+09,9E+09,9E+09,9E+09,9E+09]];
    CONST robtarget Target_870_2:=[[127.189,-1.204,10],[0,0,1,0],[0,0,-2,0],[9E+09,9E+09,9E+09,9E+09,9E+09,9E+09]];
    CONST robtarget Target_880_2:=[[115.486,8.092,10],[0,0,1,0],[0,0,-2,0],[9E+09,9E+09,9E+09,9E+09,9E+09,9E+09]];
    CONST robtarget Target_890_2:=[[115.486,17.054,10],[0,0,1,0],[0,0,-2,0],[9E+09,9E+09,9E+09,9E+09,9E+09,9E+09]];
    CONST robtarget Target_900_2:=[[127.189,17.054,10],[0,0,1,0],[0,0,-2,0],[9E+09,9E+09,9E+09,9E+09,9E+09,9E+09]];
    CONST robtarget Target_910_2:=[[138.892,17.054,10],[0,0,1,0],[0,0,-2,0],[9E+09,9E+09,9E+09,9E+09,9E+09,9E+09]];
    CONST robtarget Target_920_2:=[[138.892,24.872,10],[0,0,1,0],[0,0,-2,0],[9E+09,9E+09,9E+09,9E+09,9E+09,9E+09]];
    CONST robtarget Target_930_2:=[[109.479,24.872,10],[0,0,1,0],[0,0,-2,0],[9E+09,9E+09,9E+09,9E+09,9E+09,9E+09]];
    CONST robtarget J1_offset_2:=[[80.066,56.669,20],[0,0,1,0],[0,0,-2,0],[9E+09,9E+09,9E+09,9E+09,9E+09,9E+09]];
    CONST robtarget Target_940_2:=[[80.066,56.669,10],[0,0,1,0],[0,0,-2,0],[9E+09,9E+09,9E+09,9E+09,9E+09,9E+09]];
    CONST robtarget Target_950_2:=[[80.066,46.538,10],[0,0,1,0],[0,0,-2,0],[9E+09,9E+09,9E+09,9E+09,9E+09,9E+09]];
    CONST robtarget Target_960_2:=[[80.066,36.408,10],[0,0,1,0],[0,0,-2,0],[9E+09,9E+09,9E+09,9E+09,9E+09,9E+09]];
    CONST robtarget Target_970_2:=[[101.828,36.408,10],[0,0,1,0],[0,0,-2,0],[9E+09,9E+09,9E+09,9E+09,9E+09,9E+09]];
    CONST robtarget Target_980_2:=[[123.59,36.408,10],[0,0,1,0],[0,0,-2,0],[9E+09,9E+09,9E+09,9E+09,9E+09,9E+09]];
    CONST robtarget Target_990_2:=[[135.507,41.128,10],[0,0,1,0],[0,0,-2,0],[9E+09,9E+09,9E+09,9E+09,9E+09,9E+09]];
    CONST robtarget Target_1000_2:=[[139.702,53.809,10],[0,0,1,0],[0,0,-2,0],[9E+09,9E+09,9E+09,9E+09,9E+09,9E+09]];
    CONST robtarget Target_1010_2:=[[138.558,64.201,10],[0,0,1,0],[0,0,-2,0],[9E+09,9E+09,9E+09,9E+09,9E+09,9E+09]];
    CONST robtarget Target_1020_2:=[[131.026,63.772,10],[0,0,1,0],[0,0,-2,0],[9E+09,9E+09,9E+09,9E+09,9E+09,9E+09]];
    CONST robtarget Target_1030_2:=[[132.266,59.744,10],[0,0,1,0],[0,0,-2,0],[9E+09,9E+09,9E+09,9E+09,9E+09,9E+09]];
    CONST robtarget Target_1040_2:=[[132.933,54.857,10],[0,0,1,0],[0,0,-2,0],[9E+09,9E+09,9E+09,9E+09,9E+09,9E+09]];
    CONST robtarget Target_1050_2:=[[132.099,49.065,10],[0,0,1,0],[0,0,-2,0],[9E+09,9E+09,9E+09,9E+09,9E+09,9E+09]];
    CONST robtarget Target_1060_2:=[[129.739,45.895,10],[0,0,1,0],[0,0,-2,0],[9E+09,9E+09,9E+09,9E+09,9E+09,9E+09]];
    CONST robtarget Target_1070_2:=[[125.878,44.513,10],[0,0,1,0],[0,0,-2,0],[9E+09,9E+09,9E+09,9E+09,9E+09,9E+09]];
    CONST robtarget Target_1080_2:=[[120.586,44.227,10],[0,0,1,0],[0,0,-2,0],[9E+09,9E+09,9E+09,9E+09,9E+09,9E+09]];
    CONST robtarget Target_1090_2:=[[103.448,44.226,10],[0,0,1,0],[0,0,-2,0],[9E+09,9E+09,9E+09,9E+09,9E+09,9E+09]];
    CONST robtarget Target_1100_2:=[[86.311,44.226,10],[0,0,1,0],[0,0,-2,0],[9E+09,9E+09,9E+09,9E+09,9E+09,9E+09]];
    CONST robtarget Target_1110_2:=[[86.311,56.669,10],[0,0,1,0],[0,0,-2,0],[9E+09,9E+09,9E+09,9E+09,9E+09,9E+09]];
    CONST robtarget J2_offset_2:=[[80.065,90.372,20],[0,0,1,0],[0,0,-2,0],[9E+09,9E+09,9E+09,9E+09,9E+09,9E+09]];
    CONST robtarget Target_1120_2:=[[80.065,90.372,10],[0,0,1,0],[0,0,-2,0],[9E+09,9E+09,9E+09,9E+09,9E+09,9E+09]];
    CONST robtarget Target_1130_2:=[[80.065,80.242,10],[0,0,1,0],[0,0,-2,0],[9E+09,9E+09,9E+09,9E+09,9E+09,9E+09]];
    CONST robtarget Target_1140_2:=[[80.066,70.112,10],[0,0,1,0],[0,0,-2,0],[9E+09,9E+09,9E+09,9E+09,9E+09,9E+09]];
    CONST robtarget Target_1150_2:=[[101.827,70.112,10],[0,0,1,0],[0,0,-2,0],[9E+09,9E+09,9E+09,9E+09,9E+09,9E+09]];
    CONST robtarget Target_1160_2:=[[123.589,70.112,10],[0,0,1,0],[0,0,-2,0],[9E+09,9E+09,9E+09,9E+09,9E+09,9E+09]];
    CONST robtarget Target_1170_2:=[[135.507,74.832,10],[0,0,1,0],[0,0,-2,0],[9E+09,9E+09,9E+09,9E+09,9E+09,9E+09]];
    CONST robtarget Target_1180_2:=[[139.702,87.512,10],[0,0,1,0],[0,0,-2,0],[9E+09,9E+09,9E+09,9E+09,9E+09,9E+09]];
    CONST robtarget Target_1190_2:=[[139.369,92.589,10],[0,0,1,0],[0,0,-2,0],[9E+09,9E+09,9E+09,9E+09,9E+09,9E+09]];
    CONST robtarget Target_1200_2:=[[138.558,97.905,10],[0,0,1,0],[0,0,-2,0],[9E+09,9E+09,9E+09,9E+09,9E+09,9E+09]];
    CONST robtarget Target_1210_2:=[[134.792,97.905,10],[0,0,1,0],[0,0,-2,0],[9E+09,9E+09,9E+09,9E+09,9E+09,9E+09]];
    CONST robtarget Target_1220_2:=[[131.026,97.475,10],[0,0,1,0],[0,0,-2,0],[9E+09,9E+09,9E+09,9E+09,9E+09,9E+09]];
    CONST robtarget Target_1230_2:=[[132.265,93.447,10],[0,0,1,0],[0,0,-2,0],[9E+09,9E+09,9E+09,9E+09,9E+09,9E+09]];
    CONST robtarget Target_1240_2:=[[132.933,88.561,10],[0,0,1,0],[0,0,-2,0],[9E+09,9E+09,9E+09,9E+09,9E+09,9E+09]];
    CONST robtarget Target_1250_2:=[[132.099,82.769,10],[0,0,1,0],[0,0,-2,0],[9E+09,9E+09,9E+09,9E+09,9E+09,9E+09]];
    CONST robtarget Target_1260_2:=[[129.739,79.599,10],[0,0,1,0],[0,0,-2,0],[9E+09,9E+09,9E+09,9E+09,9E+09,9E+09]];
    CONST robtarget Target_1270_2:=[[125.878,78.216,10],[0,0,1,0],[0,0,-2,0],[9E+09,9E+09,9E+09,9E+09,9E+09,9E+09]];
    CONST robtarget Target_1280_2:=[[120.586,77.93,10],[0,0,1,0],[0,0,-2,0],[9E+09,9E+09,9E+09,9E+09,9E+09,9E+09]];
    CONST robtarget Target_1290_2:=[[110.666,78.402,10],[0,0,1,0],[0,0,-2,0],[9E+09,9E+09,9E+09,9E+09,9E+09,9E+09]];
    CONST robtarget Target_1300_2:=[[86.31,77.93,10],[0,0,1,0],[0,0,-2,0],[9E+09,9E+09,9E+09,9E+09,9E+09,9E+09]];
    CONST robtarget Target_1310_2:=[[86.31,90.372,10],[0,0,1,0],[0,0,-2,0],[9E+09,9E+09,9E+09,9E+09,9E+09,9E+09]];
    CONST robtarget Circle_offset_2:=[[-40.933895973,-5.82304871,40],[0,1,0,0],[0,0,-5,1],[9E+09,9E+09,9E+09,9E+09,9E+09,9E+09]];
    CONST robtarget Target_1330_2:=[[-40.933895973,-5.82304871,10],[0,1,0,0],[0,0,-5,1],[9E+09,9E+09,9E+09,9E+09,9E+09,9E+09]];
    CONST robtarget Target_1340_2:=[[-19.93416425,39.773116891,10],[0,1,0,0],[-1,-1,-4,1],[9E+09,9E+09,9E+09,9E+09,9E+09,9E+09]];
    CONST robtarget Target_1350_2:=[[-40.934569392,85.369917227,10],[0,1,0,0],[-1,-1,-4,1],[9E+09,9E+09,9E+09,9E+09,9E+09,9E+09]];
    CONST robtarget Target_1360_2:=[[-45.307466947,88.773192557,10],[0,1,0,0],[-1,-1,-4,1],[9E+09,9E+09,9E+09,9E+09,9E+09,9E+09]];
    CONST robtarget Target_1370_2:=[[-86.904601275,99.366718349,10],[0,1,0,0],[-1,-1,-4,1],[9E+09,9E+09,9E+09,9E+09,9E+09,9E+09]];
    CONST robtarget Target_1380_2:=[[-124.934724159,79.459035651,10],[0,1,0,0],[-1,-1,-4,1],[9E+09,9E+09,9E+09,9E+09,9E+09,9E+09]];
    CONST robtarget Target_1390_2:=[[-132.460361347,68.772867492,10],[0,1,0,0],[-1,-1,-4,1],[9E+09,9E+09,9E+09,9E+09,9E+09,9E+09]];
    CONST robtarget Target_1400_2:=[[-139.934438017,39.773268565,10],[0,1,0,0],[-1,-1,-4,1],[9E+09,9E+09,9E+09,9E+09,9E+09,9E+09]];
    CONST robtarget Target_1410_2:=[[-132.460399107,10.77239383,10],[0,1,0,0],[-1,-1,-4,1],[9E+09,9E+09,9E+09,9E+09,9E+09,9E+09]];
    CONST robtarget Target_1420_2:=[[-124.934206216,0.086767195,10],[0,1,0,0],[-1,-1,-4,1],[9E+09,9E+09,9E+09,9E+09,9E+09,9E+09]];
    CONST robtarget Target_1430_2:=[[-86.904215372,-19.820139957,10],[0,1,0,0],[0,0,-5,1],[9E+09,9E+09,9E+09,9E+09,9E+09,9E+09]];
    CONST robtarget Target_1440_2:=[[-45.307855796,-9.226362018,10],[0,1,0,0],[0,0,-5,1],[9E+09,9E+09,9E+09,9E+09,9E+09,9E+09]];
    CONST robtarget Target_1450_2:=[[-80.972940534,2.559268073,10],[0,1,0,0],[-1,-1,-4,1],[9E+09,9E+09,9E+09,9E+09,9E+09,9E+09]];
    CONST robtarget Target_1460_2:=[[-110.207862361,26.143998086,10],[0,1,0,0],[-1,-1,-4,1],[9E+09,9E+09,9E+09,9E+09,9E+09,9E+09]];
    CONST robtarget Target_1470_2:=[[-118.12963234,13.431074685,10],[0,1,0,0],[-1,-1,-4,1],[9E+09,9E+09,9E+09,9E+09,9E+09,9E+09]];
    CONST robtarget Target_1480_2:=[[-124.934206216,0.086767195,10],[0,1,0,0],[-1,-1,-4,1],[9E+09,9E+09,9E+09,9E+09,9E+09,9E+09]];
    CONST robtarget Target_1490_2:=[[-132.460399107,10.77239383,10],[0,1,0,0],[-1,-1,-4,1],[9E+09,9E+09,9E+09,9E+09,9E+09,9E+09]];
    CONST robtarget Target_1500_2:=[[-127.413721906,25.736314013,10],[0,1,0,0],[-1,-1,-4,1],[9E+09,9E+09,9E+09,9E+09,9E+09,9E+09]];
    CONST robtarget Target_1510_2:=[[-120.179725035,39.773180446,10],[0,1,0,0],[-1,-1,-4,1],[9E+09,9E+09,9E+09,9E+09,9E+09,9E+09]];
    CONST robtarget Target_1520_2:=[[-127.413036308,53.809835782,10],[0,1,0,0],[-1,-1,-4,1],[9E+09,9E+09,9E+09,9E+09,9E+09,9E+09]];
    CONST robtarget Target_1530_2:=[[-132.460361347,68.772867492,10],[0,1,0,0],[-1,-1,-4,1],[9E+09,9E+09,9E+09,9E+09,9E+09,9E+09]];
    CONST robtarget Target_1540_2:=[[-124.934724159,79.459035651,10],[0,1,0,0],[-1,-1,-4,1],[9E+09,9E+09,9E+09,9E+09,9E+09,9E+09]];
    CONST robtarget Target_1550_2:=[[-118.129234234,66.115306641,10],[0,1,0,0],[-1,-1,-4,1],[9E+09,9E+09,9E+09,9E+09,9E+09,9E+09]];
    CONST robtarget Target_1560_2:=[[-110.208779056,53.402138084,10],[0,1,0,0],[-1,-1,-4,1],[9E+09,9E+09,9E+09,9E+09,9E+09,9E+09]];
    CONST robtarget Target_1570_2:=[[-80.973561626,76.987307975,10],[0,1,0,0],[-1,-1,-4,1],[9E+09,9E+09,9E+09,9E+09,9E+09,9E+09]];
    CONST robtarget Target_1580_2:=[[-45.307466947,88.773192557,10],[0,1,0,0],[-1,-1,-4,1],[9E+09,9E+09,9E+09,9E+09,9E+09,9E+09]];
    CONST robtarget Target_1590_2:=[[-40.934569392,85.369917227,10],[0,1,0,0],[-1,-1,-4,1],[9E+09,9E+09,9E+09,9E+09,9E+09,9E+09]];
    CONST robtarget Target_1600_2:=[[-72.858424166,65.74477085,10],[0,1,0,0],[-1,-1,-4,1],[9E+09,9E+09,9E+09,9E+09,9E+09,9E+09]];
    CONST robtarget Target_1610_2:=[[-99.870719718,39.77300876,10],[0,1,0,0],[-1,-1,-4,1],[9E+09,9E+09,9E+09,9E+09,9E+09,9E+09]];
    CONST robtarget Target_1620_2:=[[-72.85802852,13.802107751,10],[0,1,0,0],[-1,-1,-4,1],[9E+09,9E+09,9E+09,9E+09,9E+09,9E+09]];
    CONST robtarget Target_1630_2:=[[-40.933895973,-5.82304871,10],[0,1,0,0],[0,0,-5,1],[9E+09,9E+09,9E+09,9E+09,9E+09,9E+09]];
    CONST robtarget Mantenimiento:=[[-440.346817367,-215.154198528,446.442364231],[0.37290991,0.812355479,0.194688267,-0.403872819],[0,0,0,0],[9E+09,9E+09,9E+09,9E+09,9E+09,9E+09]];
!***********************************************************
    !
    ! M?dulo:  Module1
    !
    ! Descripción:
    !   <Introduzca la descripción aquí>
    !
    ! Autor: Juan David
    !
    ! Versión: 1.0
    !
    !***********************************************************


    !***********************************************************
    !
    ! Procedimiento Main
    !
    !   Este es el punto de entrada de su programa
    !
    !***********************************************************
    PROC main()
        Path_Logo_30;
    ENDPROC
    PROC Path_Logo()
        MoveJ Inicio,v100,fine,TToolLab1\WObj:=Logo;
        MoveJ X1_offset,v100,fine,TToolLab1\WObj:=Logo;
        MoveL Target_10,v100,fine,TToolLab1\WObj:=Logo;
        MoveL Target_20,v100,z10,TToolLab1\WObj:=Logo;
        MoveL Target_30,v100,z10,TToolLab1\WObj:=Logo;
        MoveL Target_40,v100,z10,TToolLab1\WObj:=Logo;
        MoveL Target_50,v100,z10,TToolLab1\WObj:=Logo;
        MoveL Target_60,v100,z10,TToolLab1\WObj:=Logo;
        MoveL Target_70,v100,z10,TToolLab1\WObj:=Logo;
        MoveL Target_80,v100,z10,TToolLab1\WObj:=Logo;
        MoveL Target_90,v100,z10,TToolLab1\WObj:=Logo;
        MoveL Target_100,v100,z10,TToolLab1\WObj:=Logo;
        MoveL Target_110,v100,z10,TToolLab1\WObj:=Logo;
        MoveL Target_120,v100,z10,TToolLab1\WObj:=Logo;
        MoveL Target_130,v100,z10,TToolLab1\WObj:=Logo;
        MoveL Target_140,v100,z10,TToolLab1\WObj:=Logo;
        MoveL Target_150,v100,z10,TToolLab1\WObj:=Logo;
        MoveL Target_160,v100,z10,TToolLab1\WObj:=Logo;
        MoveL Target_170,v100,z10,TToolLab1\WObj:=Logo;
        MoveL Target_180,v100,z10,TToolLab1\WObj:=Logo;
        MoveL Target_190,v100,z10,TToolLab1\WObj:=Logo;
        MoveL Target_200,v100,z10,TToolLab1\WObj:=Logo;
        MoveL Target_10,v100,z10,TToolLab1\WObj:=Logo;
        MoveJ X1_offset,v100,z10,TToolLab1\WObj:=Logo;
        MoveJ B_offset,v100,z10,TToolLab1\WObj:=Logo;
        MoveL Target_210,v100,fine,TToolLab1\WObj:=Logo;
        MoveL Target_220,v100,z10,TToolLab1\WObj:=Logo;
        MoveL Target_230,v100,z10,TToolLab1\WObj:=Logo;
        MoveL Target_240,v100,z10,TToolLab1\WObj:=Logo;
        MoveL Target_250,v100,z10,TToolLab1\WObj:=Logo;
        MoveL Target_260,v100,z10,TToolLab1\WObj:=Logo;
        MoveL Target_270,v100,z10,TToolLab1\WObj:=Logo;
        MoveL Target_280,v100,z10,TToolLab1\WObj:=Logo;
        MoveL Target_290,v100,z10,TToolLab1\WObj:=Logo;
        MoveL Target_300,v100,z10,TToolLab1\WObj:=Logo;
        MoveL Target_310,v100,z10,TToolLab1\WObj:=Logo;
        MoveL Target_320,v100,z10,TToolLab1\WObj:=Logo;
        MoveL Target_330,v100,z10,TToolLab1\WObj:=Logo;
        MoveL Target_340,v100,z10,TToolLab1\WObj:=Logo;
        MoveL Target_350,v100,z10,TToolLab1\WObj:=Logo;
        MoveL Target_360,v100,z10,TToolLab1\WObj:=Logo;
        MoveL Target_370,v100,z10,TToolLab1\WObj:=Logo;
        MoveL Target_380,v100,z10,TToolLab1\WObj:=Logo;
        MoveL Target_210,v100,z10,TToolLab1\WObj:=Logo;
        MoveJ B_offset,v100,z10,TToolLab1\WObj:=Logo;
        MoveJ O_offset,v100,z10,TToolLab1\WObj:=Logo;
        MoveL Target_390,v100,fine,TToolLab1\WObj:=Logo;
        MoveL Target_400,v100,z10,TToolLab1\WObj:=Logo;
        MoveL Target_410,v100,z10,TToolLab1\WObj:=Logo;
        MoveL Target_420,v100,z10,TToolLab1\WObj:=Logo;
        MoveL Target_430,v100,z10,TToolLab1\WObj:=Logo;
        MoveL Target_440,v100,z10,TToolLab1\WObj:=Logo;
        MoveL Target_450,v100,z10,TToolLab1\WObj:=Logo;
        MoveL Target_460,v100,z10,TToolLab1\WObj:=Logo;
        MoveL Target_470,v100,z10,TToolLab1\WObj:=Logo;
        MoveL Target_480,v100,z10,TToolLab1\WObj:=Logo;
        MoveL Target_490,v100,z10,TToolLab1\WObj:=Logo;
        MoveL Target_500,v100,z10,TToolLab1\WObj:=Logo;
        MoveL Target_510,v100,z10,TToolLab1\WObj:=Logo;
        MoveL Target_520,v100,z10,TToolLab1\WObj:=Logo;
        MoveL Target_530,v100,z10,TToolLab1\WObj:=Logo;
        MoveL Target_540,v100,z10,TToolLab1\WObj:=Logo;
        MoveL Target_390,v100,z10,TToolLab1\WObj:=Logo;
        MoveJ O_offset,v100,z10,TToolLab1\WObj:=Logo;
        MoveJ X2_offset,v100,fine,TToolLab1\WObj:=Logo;
        MoveL Target_550,v100,fine,TToolLab1\WObj:=Logo;
        MoveL Target_560,v100,z10,TToolLab1\WObj:=Logo;
        MoveL Target_570,v100,z10,TToolLab1\WObj:=Logo;
        MoveL Target_580,v100,z10,TToolLab1\WObj:=Logo;
        MoveL Target_590,v100,z10,TToolLab1\WObj:=Logo;
        MoveL Target_600,v100,z10,TToolLab1\WObj:=Logo;
        MoveL Target_610,v100,z10,TToolLab1\WObj:=Logo;
        MoveL Target_620,v100,z10,TToolLab1\WObj:=Logo;
        MoveJ Target_630,v100,fine,TToolLab1\WObj:=Logo;
        MoveL Target_640,v100,z10,TToolLab1\WObj:=Logo;
        MoveL Target_650,v100,z10,TToolLab1\WObj:=Logo;
        MoveL Target_660,v100,z10,TToolLab1\WObj:=Logo;
        MoveL Target_670,v100,z10,TToolLab1\WObj:=Logo;
        MoveL Target_680,v100,z10,TToolLab1\WObj:=Logo;
        MoveL Target_690,v100,z10,TToolLab1\WObj:=Logo;
        MoveL Target_700,v100,z10,TToolLab1\WObj:=Logo;
        MoveL Target_710,v100,z10,TToolLab1\WObj:=Logo;
        MoveL Target_720,v100,z10,TToolLab1\WObj:=Logo;
        MoveL Target_730,v100,z10,TToolLab1\WObj:=Logo;
        MoveL Target_740,v100,z10,TToolLab1\WObj:=Logo;
        MoveL Target_550,v100,z10,TToolLab1\WObj:=Logo;
        MoveJ X2_offset,v100,z10,TToolLab1\WObj:=Logo;
        MoveJ R_offset,v100,fine,TToolLab1\WObj:=Logo;
        MoveL Target_750,v100,fine,TToolLab1\WObj:=Logo;
        MoveL Target_760,v100,z10,TToolLab1\WObj:=Logo;
        MoveL Target_770,v100,z10,TToolLab1\WObj:=Logo;
        MoveL Target_780,v100,z10,TToolLab1\WObj:=Logo;
        MoveL Target_790,v100,z10,TToolLab1\WObj:=Logo;
        MoveL Target_800,v100,z10,TToolLab1\WObj:=Logo;
        MoveL Target_810,v100,z10,TToolLab1\WObj:=Logo;
        MoveL Target_820,v100,z10,TToolLab1\WObj:=Logo;
        MoveL Target_830,v100,z10,TToolLab1\WObj:=Logo;
        MoveL Target_840,v100,z10,TToolLab1\WObj:=Logo;
        MoveL Target_850,v100,z10,TToolLab1\WObj:=Logo;
        MoveL Target_860,v100,z10,TToolLab1\WObj:=Logo;
        MoveL Target_870,v100,z10,TToolLab1\WObj:=Logo;
        MoveL Target_880,v100,z10,TToolLab1\WObj:=Logo;
        MoveL Target_890,v100,z10,TToolLab1\WObj:=Logo;
        MoveL Target_900,v100,z10,TToolLab1\WObj:=Logo;
        MoveL Target_910,v100,z10,TToolLab1\WObj:=Logo;
        MoveL Target_920,v100,z10,TToolLab1\WObj:=Logo;
        MoveL Target_930,v100,z10,TToolLab1\WObj:=Logo;
        MoveL Target_750,v100,z10,TToolLab1\WObj:=Logo;
        MoveJ R_offset,v100,z10,TToolLab1\WObj:=Logo;
        MoveJ J1_offset,v100,z10,TToolLab1\WObj:=Logo;
        MoveL Target_940,v100,fine,TToolLab1\WObj:=Logo;
        MoveL Target_950,v100,z10,TToolLab1\WObj:=Logo;
        MoveL Target_960,v100,z10,TToolLab1\WObj:=Logo;
        MoveL Target_970,v100,z10,TToolLab1\WObj:=Logo;
        MoveL Target_980,v100,z10,TToolLab1\WObj:=Logo;
        MoveL Target_990,v100,z10,TToolLab1\WObj:=Logo;
        MoveL Target_1000,v100,z10,TToolLab1\WObj:=Logo;
        MoveL Target_1010,v100,z10,TToolLab1\WObj:=Logo;
        MoveL Target_1020,v100,z10,TToolLab1\WObj:=Logo;
        MoveL Target_1030,v100,z10,TToolLab1\WObj:=Logo;
        MoveL Target_1040,v100,z10,TToolLab1\WObj:=Logo;
        MoveL Target_1050,v100,z10,TToolLab1\WObj:=Logo;
        MoveL Target_1060,v100,z10,TToolLab1\WObj:=Logo;
        MoveL Target_1070,v100,z10,TToolLab1\WObj:=Logo;
        MoveL Target_1080,v100,z10,TToolLab1\WObj:=Logo;
        MoveL Target_1090,v100,z10,TToolLab1\WObj:=Logo;
        MoveL Target_1100,v100,z10,TToolLab1\WObj:=Logo;
        MoveL Target_1110,v100,z10,TToolLab1\WObj:=Logo;
        MoveL Target_940,v100,z10,TToolLab1\WObj:=Logo;
        MoveJ J1_offset,v100,z10,TToolLab1\WObj:=Logo;
        MoveJ J2_offset,v100,z10,TToolLab1\WObj:=Logo;
        MoveL Target_1120,v100,fine,TToolLab1\WObj:=Logo;
        MoveL Target_1130,v100,z10,TToolLab1\WObj:=Logo;
        MoveL Target_1140,v100,z10,TToolLab1\WObj:=Logo;
        MoveL Target_1150,v100,z10,TToolLab1\WObj:=Logo;
        MoveL Target_1160,v100,z10,TToolLab1\WObj:=Logo;
        MoveL Target_1170,v100,z10,TToolLab1\WObj:=Logo;
        MoveL Target_1180,v100,z10,TToolLab1\WObj:=Logo;
        MoveL Target_1190,v100,z10,TToolLab1\WObj:=Logo;
        MoveL Target_1200,v100,z10,TToolLab1\WObj:=Logo;
        MoveL Target_1210,v100,z10,TToolLab1\WObj:=Logo;
        MoveL Target_1220,v100,z10,TToolLab1\WObj:=Logo;
        MoveL Target_1230,v100,z10,TToolLab1\WObj:=Logo;
        MoveL Target_1240,v100,z10,TToolLab1\WObj:=Logo;
        MoveL Target_1250,v100,z10,TToolLab1\WObj:=Logo;
        MoveL Target_1260,v100,z10,TToolLab1\WObj:=Logo;
        MoveL Target_1270,v100,z10,TToolLab1\WObj:=Logo;
        MoveL Target_1280,v100,z10,TToolLab1\WObj:=Logo;
        MoveL Target_1290,v100,z10,TToolLab1\WObj:=Logo;
        MoveL Target_1300,v100,z10,TToolLab1\WObj:=Logo;
        MoveL Target_1310,v100,z10,TToolLab1\WObj:=Logo;
        MoveL Target_1120,v100,z10,TToolLab1\WObj:=Logo;
        MoveJ J2_offset,v100,z10,TToolLab1\WObj:=Logo;
        MoveJ Inicio,v100,fine,TToolLab1\WObj:=Logo;
    ENDPROC
    PROC Path_Logo_30()
        WaitDI DI_1,1;
        SetDO DO_1,1;
        MoveJ Inicio,v100,z10,TToolLab1\WObj:=Logo;
        MoveJ X1_offset_2,v100,fine,TToolLab1\WObj:=Logo30;
        MoveL Target_10_2,v100,z10,TToolLab1\WObj:=Logo30;
        MoveL Target_20_2,v100,z10,TToolLab1\WObj:=Logo30;
        MoveL Target_30_2,v100,z10,TToolLab1\WObj:=Logo30;
        MoveL Target_40_2,v100,z10,TToolLab1\WObj:=Logo30;
        MoveL Target_50_2,v100,z10,TToolLab1\WObj:=Logo30;
        MoveL Target_60_2,v100,z10,TToolLab1\WObj:=Logo30;
        MoveL Target_70_2,v100,z10,TToolLab1\WObj:=Logo30;
        MoveL Target_80_2,v100,z10,TToolLab1\WObj:=Logo30;
        MoveL Target_90_2,v100,z10,TToolLab1\WObj:=Logo30;
        MoveL Target_100_2,v100,z10,TToolLab1\WObj:=Logo30;
        MoveL Target_110_2,v100,z10,TToolLab1\WObj:=Logo30;
        MoveL Target_120_2,v100,z10,TToolLab1\WObj:=Logo30;
        MoveL Target_130_2,v100,z10,TToolLab1\WObj:=Logo30;
        MoveL Target_140_2,v100,z10,TToolLab1\WObj:=Logo30;
        MoveL Target_150_2,v100,z10,TToolLab1\WObj:=Logo30;
        MoveL Target_160_2,v100,z10,TToolLab1\WObj:=Logo30;
        MoveL Target_170_2,v100,z10,TToolLab1\WObj:=Logo30;
        MoveL Target_180_2,v100,z10,TToolLab1\WObj:=Logo30;
        MoveL Target_190_2,v100,z10,TToolLab1\WObj:=Logo30;
        MoveL Target_200_2,v100,z10,TToolLab1\WObj:=Logo30;
        MoveL Target_10_2,v100,z10,TToolLab1\WObj:=Logo30;
        MoveJ X1_offset_2,v100,fine,TToolLab1\WObj:=Logo30;
        MoveJ B_offset_2,v100,fine,TToolLab1\WObj:=Logo30;
        MoveL Target_210_2,v100,z10,TToolLab1\WObj:=Logo30;
        MoveL Target_220_2,v100,z10,TToolLab1\WObj:=Logo30;
        MoveL Target_230_2,v100,z10,TToolLab1\WObj:=Logo30;
        MoveL Target_240_2,v100,z10,TToolLab1\WObj:=Logo30;
        MoveL Target_250_2,v100,z10,TToolLab1\WObj:=Logo30;
        MoveL Target_260_2,v100,z10,TToolLab1\WObj:=Logo30;
        MoveL Target_270_2,v100,z10,TToolLab1\WObj:=Logo30;
        MoveL Target_280_2,v100,z10,TToolLab1\WObj:=Logo30;
        MoveL Target_290_2,v100,z10,TToolLab1\WObj:=Logo30;
        MoveL Target_300_2,v100,z10,TToolLab1\WObj:=Logo30;
        MoveL Target_310_2,v100,z10,TToolLab1\WObj:=Logo30;
        MoveL Target_320_2,v100,z10,TToolLab1\WObj:=Logo30;
        MoveL Target_330_2,v100,z10,TToolLab1\WObj:=Logo30;
        MoveL Target_340_2,v100,z10,TToolLab1\WObj:=Logo30;
        MoveL Target_350_2,v100,z10,TToolLab1\WObj:=Logo30;
        MoveL Target_360_2,v100,z10,TToolLab1\WObj:=Logo30;
        MoveL Target_370_2,v100,z10,TToolLab1\WObj:=Logo30;
        MoveL Target_380_2,v100,z10,TToolLab1\WObj:=Logo30;
        MoveL Target_210_2,v100,z10,TToolLab1\WObj:=Logo30;
        MoveJ B_offset_2,v100,fine,TToolLab1\WObj:=Logo30;
        MoveJ O_offset_2,v100,fine,TToolLab1\WObj:=Logo30;
        MoveL Target_390_2,v100,z10,TToolLab1\WObj:=Logo30;
        MoveL Target_400_2,v100,z10,TToolLab1\WObj:=Logo30;
        MoveL Target_410_2,v100,z10,TToolLab1\WObj:=Logo30;
        MoveL Target_420_2,v100,z10,TToolLab1\WObj:=Logo30;
        MoveL Target_430_2,v100,z10,TToolLab1\WObj:=Logo30;
        MoveL Target_440_2,v100,z10,TToolLab1\WObj:=Logo30;
        MoveL Target_450_2,v100,z10,TToolLab1\WObj:=Logo30;
        MoveL Target_460_2,v100,z10,TToolLab1\WObj:=Logo30;
        MoveL Target_470_2,v100,z10,TToolLab1\WObj:=Logo30;
        MoveL Target_480_2,v100,z10,TToolLab1\WObj:=Logo30;
        MoveL Target_490_2,v100,z10,TToolLab1\WObj:=Logo30;
        MoveL Target_500_2,v100,z10,TToolLab1\WObj:=Logo30;
        MoveL Target_510_2,v100,z10,TToolLab1\WObj:=Logo30;
        MoveL Target_520_2,v100,z10,TToolLab1\WObj:=Logo30;
        MoveL Target_530_2,v100,z10,TToolLab1\WObj:=Logo30;
        MoveL Target_540_2,v100,z10,TToolLab1\WObj:=Logo30;
        MoveL Target_390_2,v100,z10,TToolLab1\WObj:=Logo30;
        MoveJ O_offset_2,v100,fine,TToolLab1\WObj:=Logo30;
        MoveJ X2_offset_2,v100,fine,TToolLab1\WObj:=Logo30;
        MoveL Target_550_2,v100,z10,TToolLab1\WObj:=Logo30;
        MoveL Target_560_2,v100,z10,TToolLab1\WObj:=Logo30;
        MoveL Target_570_2,v100,z10,TToolLab1\WObj:=Logo30;
        MoveL Target_580_2,v100,z10,TToolLab1\WObj:=Logo30;
        MoveL Target_590_2,v100,z10,TToolLab1\WObj:=Logo30;
        MoveL Target_600_2,v100,z10,TToolLab1\WObj:=Logo30;
        MoveL Target_610_2,v100,z10,TToolLab1\WObj:=Logo30;
        MoveL Target_620_2,v100,z10,TToolLab1\WObj:=Logo30;
        MoveL Target_630_2,v100,z10,TToolLab1\WObj:=Logo30;
        MoveL Target_640_2,v100,z10,TToolLab1\WObj:=Logo30;
        MoveL Target_650_2,v100,z10,TToolLab1\WObj:=Logo30;
        MoveL Target_660_2,v100,z10,TToolLab1\WObj:=Logo30;
        MoveL Target_670_2,v100,z10,TToolLab1\WObj:=Logo30;
        MoveL Target_680_2,v100,z10,TToolLab1\WObj:=Logo30;
        MoveL Target_690_2,v100,z10,TToolLab1\WObj:=Logo30;
        MoveL Target_700_2,v100,z10,TToolLab1\WObj:=Logo30;
        MoveL Target_710_2,v100,z10,TToolLab1\WObj:=Logo30;
        MoveL Target_720_2,v100,z10,TToolLab1\WObj:=Logo30;
        MoveL Target_730_2,v100,z10,TToolLab1\WObj:=Logo30;
        MoveL Target_740_2,v100,z10,TToolLab1\WObj:=Logo30;
        MoveL Target_550_2,v100,z10,TToolLab1\WObj:=Logo30;
        MoveJ X2_offset_2,v100,fine,TToolLab1\WObj:=Logo30;
        MoveJ R_offset_2,v100,fine,TToolLab1\WObj:=Logo30;
        MoveL Target_750_2,v100,fine,TToolLab1\WObj:=Logo30;
        MoveL Target_760_2,v100,fine,TToolLab1\WObj:=Logo30;
        MoveL Target_770_2,v100,fine,TToolLab1\WObj:=Logo30;
        MoveL Target_780_2,v100,fine,TToolLab1\WObj:=Logo30;
        MoveL Target_790_2,v100,fine,TToolLab1\WObj:=Logo30;
        MoveL Target_800_2,v100,fine,TToolLab1\WObj:=Logo30;
        MoveL Target_810_2,v100,fine,TToolLab1\WObj:=Logo30;
        MoveL Target_820_2,v100,fine,TToolLab1\WObj:=Logo30;
        MoveL Target_830_2,v100,fine,TToolLab1\WObj:=Logo30;
        MoveL Target_840_2,v100,fine,TToolLab1\WObj:=Logo30;
        MoveL Target_850_2,v100,fine,TToolLab1\WObj:=Logo30;
        MoveL Target_860_2,v100,fine,TToolLab1\WObj:=Logo30;
        MoveL Target_870_2,v100,fine,TToolLab1\WObj:=Logo30;
        MoveL Target_880_2,v100,fine,TToolLab1\WObj:=Logo30;
        MoveL Target_890_2,v100,fine,TToolLab1\WObj:=Logo30;
        MoveL Target_900_2,v100,fine,TToolLab1\WObj:=Logo30;
        MoveL Target_910_2,v100,fine,TToolLab1\WObj:=Logo30;
        MoveL Target_920_2,v100,fine,TToolLab1\WObj:=Logo30;
        MoveL Target_930_2,v100,fine,TToolLab1\WObj:=Logo30;
        MoveL Target_750_2,v100,fine,TToolLab1\WObj:=Logo30;
        MoveJ R_offset_2,v100,fine,TToolLab1\WObj:=Logo30;
        MoveJ J1_offset_2,v100,fine,TToolLab1\WObj:=Logo30;
        MoveL Target_940_2,v100,z10,TToolLab1\WObj:=Logo30;
        MoveL Target_950_2,v100,z10,TToolLab1\WObj:=Logo30;
        MoveL Target_960_2,v100,z10,TToolLab1\WObj:=Logo30;
        MoveL Target_970_2,v100,z10,TToolLab1\WObj:=Logo30;
        MoveL Target_980_2,v100,z10,TToolLab1\WObj:=Logo30;
        MoveL Target_990_2,v100,z10,TToolLab1\WObj:=Logo30;
        MoveL Target_1000_2,v100,z10,TToolLab1\WObj:=Logo30;
        MoveL Target_1010_2,v100,z10,TToolLab1\WObj:=Logo30;
        MoveL Target_1020_2,v100,z10,TToolLab1\WObj:=Logo30;
        MoveL Target_1030_2,v100,z10,TToolLab1\WObj:=Logo30;
        MoveL Target_1040_2,v100,z10,TToolLab1\WObj:=Logo30;
        MoveL Target_1050_2,v100,z10,TToolLab1\WObj:=Logo30;
        MoveL Target_1060_2,v100,z10,TToolLab1\WObj:=Logo30;
        MoveL Target_1070_2,v100,z10,TToolLab1\WObj:=Logo30;
        MoveL Target_1080_2,v100,z10,TToolLab1\WObj:=Logo30;
        MoveL Target_1090_2,v100,z10,TToolLab1\WObj:=Logo30;
        MoveL Target_1100_2,v100,z10,TToolLab1\WObj:=Logo30;
        MoveL Target_1110_2,v100,z10,TToolLab1\WObj:=Logo30;
        MoveL Target_940_2,v100,z10,TToolLab1\WObj:=Logo30;
        MoveJ J1_offset_2,v100,fine,TToolLab1\WObj:=Logo30;
        MoveJ J2_offset_2,v100,fine,TToolLab1\WObj:=Logo30;
        MoveL Target_1120_2,v100,fine,TToolLab1\WObj:=Logo30;
        MoveL Target_1130_2,v100,fine,TToolLab1\WObj:=Logo30;
        MoveL Target_1140_2,v100,fine,TToolLab1\WObj:=Logo30;
        MoveL Target_1150_2,v100,fine,TToolLab1\WObj:=Logo30;
        MoveL Target_1160_2,v100,fine,TToolLab1\WObj:=Logo30;
        MoveL Target_1170_2,v100,fine,TToolLab1\WObj:=Logo30;
        MoveL Target_1180_2,v100,fine,TToolLab1\WObj:=Logo30;
        MoveL Target_1190_2,v100,fine,TToolLab1\WObj:=Logo30;
        MoveL Target_1200_2,v100,fine,TToolLab1\WObj:=Logo30;
        MoveL Target_1210_2,v100,fine,TToolLab1\WObj:=Logo30;
        MoveL Target_1220_2,v100,fine,TToolLab1\WObj:=Logo30;
        MoveL Target_1230_2,v100,fine,TToolLab1\WObj:=Logo30;
        MoveL Target_1240_2,v100,fine,TToolLab1\WObj:=Logo30;
        MoveL Target_1250_2,v100,fine,TToolLab1\WObj:=Logo30;
        MoveL Target_1260_2,v100,fine,TToolLab1\WObj:=Logo30;
        MoveL Target_1270_2,v100,fine,TToolLab1\WObj:=Logo30;
        MoveL Target_1280_2,v100,fine,TToolLab1\WObj:=Logo30;
        MoveL Target_1290_2,v100,fine,TToolLab1\WObj:=Logo30;
        MoveL Target_1300_2,v100,fine,TToolLab1\WObj:=Logo30;
        MoveL Target_1310_2,v100,fine,TToolLab1\WObj:=Logo30;
        MoveL Target_1120_2,v100,z10,TToolLab1\WObj:=Logo30;
        MoveJ J2_offset_2,v100,fine,TToolLab1\WObj:=Logo30;
        MoveJ Inicio,v100,z10,TToolLab1\WObj:=Logo;
        WaitDI DI_2,1;
        Path_Mantenimiento;
    ENDPROC
    PROC Path_Mantenimiento()
        SetDO DO_1,0;
        MoveJ Mantenimiento,v100,fine,TToolLab1\WObj:=Logo30;
    ENDPROC
ENDMODULE
